{attribute 'linkalways'} 
{attribute 'no_explicit_call' := 'This FB is a CLASS and must be accessed using methods or properties'}
{attribute 'enable_dynamic_creation'}
FUNCTION_BLOCK FINAL GE_SINT EXTENDS Node
VAR
	in1 : _SINT(0);
	in2 : _SINT(0);
	out : _BOOL(FALSE);
END_VAR

METHOD PUBLIC Clone : I_Node
VAR
	pNode : POINTER TO GE_SINT;
END_VAR
pNode := __NEW(GE_SINT);
Clone := pNode^;
END_METHOD

METHOD FB_init : BOOL
VAR_INPUT
	bInitRetains : BOOL; // if TRUE, the retain variables are initialized (warm start / cold start)
	bInCopyCode : BOOL;  // if TRUE, the instance afterwards gets moved into the copy code (online change)
END_VAR
AddInput('in1',THIS^.in1);
AddInput('in2',THIS^.in2);
AddOutput('out', THIS^.out);
END_METHOD

METHOD PROTECTED OnExecute
VAR
END_VAR
out.Value := in1.Value >= in2.Value;
END_METHOD

END_FUNCTION_BLOCK

(* stored: Version 1.1.0.1, ProductVersion 3.1.4024.15
   POU GE_SINT: Id {b039e070-e536-49aa-b50a-a9677d6ef1c6}, SpecialFunc None
   Folder Constructor: Id {8f1f11e5-eaac-4b61-80af-928cf6904e80}
   Method Clone: Id {0e2a13e2-fb72-4440-ade4-f49edc71186a}
   Method FB_init: Id {f57e22f7-1d86-42ab-999c-1c9a13c0703d}
   Method OnExecute: Id {401578af-3c6d-487d-85e2-8bf1b3e3a14a} *)
